# EPICS substitutions: rknmntrSup/test_block_curr_PVs.substitutions
file test_block_curr_PVs.template {
    pattern { MAGNET }

    { "RQ1" }
    { "RQ2" }
    { "RB1" }
}
